PROGRAM prgVarEffIO
VAR
	fbVar		: FB_VarInfo_V3;
END_VAR

fbVar(
	bReadInfo:= , 
	eTMCFile:= eSelectTMCFile.eDontUseTMCFile, 
	eSavePositionTMCFile:= eSavePositionOnPLC.ePostionC, 
	udiCounterFoundVariables=> , 
	bError=> , 
	bBusy=> , 
	byProgress=> , 
	udiErrorCodeOut=> , 
	eErrorVarInfo_Out=> , 
	sVarWithError=> );

fbVar(
	bReadInfo:= , 
	eTMCFile:= eSelectTMCFile.eDontUseTMCFile, 
	eSavePositionTMCFile:= eSavePositionOnPLC.ePostionC,
	udiCounterFoundVariables=> , 
	bError=> , 
	bBusy=> , 
	byProgress=> , 
	udiErrorCodeOut=> , 
	eErrorVarInfo_Out=> , 
	sVarWithError=> );
	
fbVar(
	bReadInfo:= , 
	eTMCFile:= eSelectTMCFile.eDontUseTMCFile, 
	eSavePositionTMCFile:= eSavePositionOnPLC.ePostionC,
	udiCounterFoundVariables=> , 
	bError=> , 
	bBusy=> , 
	byProgress=> , 
	udiErrorCodeOut=> , 
	eErrorVarInfo_Out=> , 
	sVarWithError=> );

END_PROGRAM

(* stored: Version 1.1.0.1, ProductVersion 3.1.4024.12
   POU prgVarEffIO: Id {688c9479-e6ec-42dd-a7ff-f4574a13d605}, SpecialFunc None *)
